Staubli VAL3: example.pgx

program example()
  local string l_sLanguage
begin
  //-----------------------------------------------------------------------
  //Header begin
  //Description of program
  //  This is an example of use of this library
  //  This program uses the following sub-programs :
  //  - language(): choose the language : "English", "French", "Spanish"
  //  - mainCalcToolpp(): calculates the tool transformation : a wizard will
  //  guide you thtough the steps.
  //History
  //  Creation : 08-04-08 - f.Rob
  //Header end
  //-----------------------------------------------------------------------

  //for choose the language
  call language(l_sLanguage)
  call mainCalcToolpp(l_sLanguage,tTool)
end
